Staubli VAL3: changeToolMove.pgx

public program changeToolMove(num nChange (dimensions=1))
begin
  call external:oGripCmd2(nChange)
end
